// TIA Portal V17 program export: 7 tag tables, 61 data types, 15 data blocks, 115 code blocks (in call order from the OBs), 16 instance data blocks

VAR_GLOBAL   // PLC tag table "Auxiliary_IO"
   Rack2Slot20_I AT %I310.0 : "stET200AL_AQ_I";   //    {ExternalAccessible false, ExternalVisible false, ExternalWritable false}
   Rack2Slot21_I AT %I320.0 : "stET200AL_AI";   //    {ExternalAccessible false, ExternalVisible false, ExternalWritable false}
   Rack1Slot9_I AT %I170.0 : "stET200AL_AI";   //    {ExternalAccessible false, ExternalVisible false, ExternalWritable false}
   Rack1Slot8_I AT %I160.0 : "stET200AL_AI";   //    {ExternalAccessible false, ExternalVisible false, ExternalWritable false}
   Rack1Slot7_I AT %I150.0 : "stET200AL_AI";   //    {ExternalAccessible false, ExternalVisible false, ExternalWritable false}
   Rack2Slot25_I AT %I360.0 : "stET200AL_AI";   //    {ExternalAccessible false, ExternalVisible false, ExternalWritable false}
   Rack1Slot5_I AT %I130.0 : "stET200AL_AI";   //    {ExternalAccessible false, ExternalVisible false, ExternalWritable false}
   Rack1Slot4_I AT %I120.0 : "stET200AL_RTD";   //    {ExternalAccessible false, ExternalVisible false, ExternalWritable false}
   Rack1Slot6_I AT %I140.0 : "stET200AL_AI";   //    {ExternalAccessible false, ExternalVisible false, ExternalWritable false}
   Rack2Slot19_I AT %I300.0 : "stET200AL_AI";   //    {ExternalAccessible false, ExternalVisible false, ExternalWritable false}
   Rack1Slot2_I AT %I100.0 : "stET200AL_AI";   //    {ExternalAccessible false, ExternalVisible false, ExternalWritable false}
   Rack2Slot23_I AT %I340.0 : "stET200AL_AI";   //    {ExternalAccessible false, ExternalVisible false, ExternalWritable false}
   Rack2Slot22_I AT %I330.0 : "stET200AL_AI";   //    {ExternalAccessible false, ExternalVisible false, ExternalWritable false}
   Rack1Slot3_I AT %I110.0 : "stET200AL_RTD";   //    {ExternalAccessible false, ExternalVisible false, ExternalWritable false}
   Rack2Slot24_I AT %I350.0 : "stET200AL_AI";   //    {ExternalAccessible false, ExternalVisible false, ExternalWritable false}
   Rack2Slot29_I AT %I400.0 : "stET200AL_AI";   //    {ExternalAccessible false, ExternalVisible false, ExternalWritable false}
   Rack2Slot30_I AT %I410.0 : "stET200AL_AI";   //    {ExternalAccessible false, ExternalVisible false, ExternalWritable false}
   Rack2Slot31_I AT %I420.0 : "stET200AL_AI";   //    {ExternalAccessible false, ExternalVisible false, ExternalWritable false}
   Rack2Slot32_I AT %I430.0 : "stET200AL_RTD";   //    {ExternalAccessible false, ExternalVisible false, ExternalWritable false}
   Rack2Slot33_I AT %I440.0 : "stET200AL_AI";   //    {ExternalAccessible false, ExternalVisible false, ExternalWritable false}
   Rack2Slot34_I AT %I450.0 : "stET200AL_AI";   //    {ExternalAccessible false, ExternalVisible false, ExternalWritable false}
   Rack2Slot26_I AT %I370.0 : "stET200AL_AQ_I";   //    {ExternalAccessible false, ExternalVisible false, ExternalWritable false}
   Rack2Slot27_I AT %I380.0 : "stET200AL_AI";   //    {ExternalAccessible false, ExternalVisible false, ExternalWritable false}
   Rack2Slot28_I AT %I390.0 : "stET200AL_AQ_I";   //    {ExternalAccessible false, ExternalVisible false, ExternalWritable false}
   Rack2Slot20_Q AT %Q310.0 : "stET200AL_AQ";   //    {ExternalAccessible false, ExternalVisible false, ExternalWritable false}
   Rack2Slot21_Q AT %Q320.0 : "stET200AL_AQ";   //    {ExternalAccessible false, ExternalVisible false, ExternalWritable false}
   Rack1Slot10_I AT %I180.0 : "stET200AL_DIQ_I";   //    {ExternalAccessible false, ExternalVisible false, ExternalWritable false}
   Rack1Slot11_I AT %I190.0 : "stET200AL_RTD";   //    {ExternalAccessible false, ExternalVisible false, ExternalWritable false}
   Rack1Slot12_I AT %I200.0 : "stET200AL_AI";   //    {ExternalAccessible false, ExternalVisible false, ExternalWritable false}
   Rack1Slot13_I AT %I210.0 : "stET200AL_AI";   //    {ExternalAccessible false, ExternalVisible false, ExternalWritable false}
   Rack1Slot14_I AT %I248.0 : "stET200AL_RTD";   //    {ExternalAccessible false, ExternalVisible false, ExternalWritable false}
   Rack1Slot15_I AT %I230.0 : "stET200AL_AI";   //    {ExternalAccessible false, ExternalVisible false, ExternalWritable false}
   Rack1Slot16_I AT %I240.0 : "stET200AL_AI";   //    {ExternalAccessible false, ExternalVisible false, ExternalWritable false}
   Rack1Slot17_I AT %I250.0 : "stET200AL_AI";   //    {ExternalAccessible false, ExternalVisible false, ExternalWritable false}
   Rack2Slot19_Q AT %Q300.0 : "stET200AL_AQ";   //    {ExternalAccessible false, ExternalVisible false, ExternalWritable false}
   Rack2Slot22_Q AT %Q330.0 : "stET200AL_AQ";   //    {ExternalAccessible false, ExternalVisible false, ExternalWritable false}
   Rack2Slot23_Q AT %Q340.0 : "stET200AL_AQ";   //    {ExternalAccessible false, ExternalVisible false, ExternalWritable false}
   Rack2Slot24_Q AT %Q350.0 : "stET200AL_AQ";   //    {ExternalAccessible false, ExternalVisible false, ExternalWritable false}
   Rack2Slot25_Q AT %Q360.0 : "stET200AL_AQ";   //    {ExternalAccessible false, ExternalVisible false, ExternalWritable false}
   Rack2Slot26_Q AT %Q370.0 : "stET200AL_AQ";   //    {ExternalAccessible false, ExternalVisible false, ExternalWritable false}
   Rack2Slot27_Q AT %Q380.0 : "stET200AL_AQ";   //    {ExternalAccessible false, ExternalVisible false, ExternalWritable false}
   Rack2Slot28_Q AT %Q390.0 : "stET200AL_AQ";   //    {ExternalAccessible false, ExternalVisible false, ExternalWritable false}
   Rack2Slot29_Q AT %Q400.0 : "stET200AL_AQ";   //    {ExternalAccessible false, ExternalVisible false, ExternalWritable false}
   Rack2Slot30_Q AT %Q410.0 : "stET200AL_AQ";   //    {ExternalAccessible false, ExternalVisible false, ExternalWritable false}
   Rack2Slot31_Q AT %Q420.0 : "stET200AL_AQ";   //    {ExternalAccessible false, ExternalVisible false, ExternalWritable false}
   Rack2Slot32_Q AT %Q430.0 : "stET200AL_AQ";   //    {ExternalAccessible false, ExternalVisible false, ExternalWritable false}
   Rack2Slot33_Q AT %Q440.0 : "stET200AL_AQ";   //    {ExternalAccessible false, ExternalVisible false, ExternalWritable false}
   Rack2Slot34_Q AT %Q450.0 : "stET200AL_AQ";   //    {ExternalAccessible false, ExternalVisible false, ExternalWritable false}
   Rack1Slot10_Q AT %Q180.0 : "stET200AL_DIQ_Q";   //    {ExternalAccessible false, ExternalVisible false, ExternalWritable false}
END_VAR

VAR_GLOBAL   // PLC tag table "Default tag table"
   Trial AT %I0.0 : Bool;
END_VAR

VAR_GLOBAL   // PLC tag table "Inverters"
   TA1_Rx AT %I10.0 : "stABB_ACSx80_Rx";   // HBL-SC-01   {ExternalAccessible false, ExternalVisible false, ExternalWritable false}
   TA1_Tx AT %Q10.0 : "stABB_ACSx80_Tx";   // HBL-SC-01   {ExternalAccessible false, ExternalVisible false, ExternalWritable false}
   TA2_Rx AT %I30.0 : "stABB_ACSx80_Rx";   // HBL-SC-02   {ExternalAccessible false, ExternalVisible false, ExternalWritable false}
   TA10_Rx AT %I68.0 : "stABB_ACSx80_Rx";   // HBL-SC-10   {ExternalAccessible false, ExternalVisible false, ExternalWritable false}
   TA2_Tx AT %Q30.0 : "stABB_ACSx80_Tx";   // HBL-SC-02   {ExternalAccessible false, ExternalVisible false, ExternalWritable false}
   TA10_Tx AT %Q68.0 : "stABB_ACSx80_Tx";   // '   {ExternalAccessible false, ExternalVisible false, ExternalWritable false}
   TA_State AT %IB7 : Byte;   // 1 = online   {ExternalAccessible false, ExternalVisible false, ExternalWritable false}
   TA3_Rx AT %I228.0 : "stABB_ACSx80_Rx";   // HBL-SC-03   {ExternalAccessible false, ExternalVisible false, ExternalWritable false}
   TA3_Tx AT %Q88.0 : "stABB_ACSx80_Tx";   // HBL-SC-03   {ExternalAccessible false, ExternalVisible false, ExternalWritable false}
END_VAR

VAR_GLOBAL   // PLC tag table "Local_IO"
   SM1222_DO_0 AT %Q8.0 : Bool;   //    {ExternalAccessible false, ExternalVisible false, ExternalWritable false}
   SM1222_DO_1 AT %Q8.1 : Bool;   //    {ExternalAccessible false, ExternalVisible false, ExternalWritable false}
   SM1222_DO_2 AT %Q8.2 : Bool;   //    {ExternalAccessible false, ExternalVisible false, ExternalWritable false}
   SM1222_DO_3 AT %Q8.3 : Bool;   //    {ExternalAccessible false, ExternalVisible false, ExternalWritable false}
   SM1222_DO_4 AT %Q8.4 : Bool;   //    {ExternalAccessible false, ExternalVisible false, ExternalWritable false}
   SM1222_DO_5 AT %Q8.5 : Bool;   //    {ExternalAccessible false, ExternalVisible false, ExternalWritable false}
   SM1222_DO_6 AT %Q8.6 : Bool;   //    {ExternalAccessible false, ExternalVisible false, ExternalWritable false}
   SM1222_DO_7 AT %Q8.7 : Bool;   //    {ExternalAccessible false, ExternalVisible false, ExternalWritable false}
   SM531 AT %I500.0 : "stSM531_4AI";   //    {ExternalAccessible false, ExternalVisible false, ExternalWritable false}
   SM521 AT %I510.0 : "stSM521_16DI";   //    {ExternalAccessible false, ExternalVisible false, ExternalWritable false}
   SM522_I AT %I512.0 : "stSM522_32DQ_I";   //    {ExternalAccessible false, ExternalVisible false, ExternalWritable false}
   SM522_Q AT %Q512.0 : "stSM522_32DQ_Q";   //    {ExternalAccessible false, ExternalVisible false, ExternalWritable false}
END_VAR

VAR_GLOBAL   // PLC tag table "RIO1"
   RIO1_Slot4_I AT %I634.0 : "stSM531_8AI";   //    {ExternalAccessible false, ExternalVisible false, ExternalWritable false}
   RIO1_Slot2_I AT %I600.0 : "stSM531_8AI";   //    {ExternalAccessible false, ExternalVisible false, ExternalWritable false}
   RIO1_Slot3_I AT %I617.0 : "stSM531_8AI";   //    {ExternalAccessible false, ExternalVisible false, ExternalWritable false}
   RIO1_Slot5_I AT %I651.0 : "stSM531_8AI";   //    {ExternalAccessible false, ExternalVisible false, ExternalWritable false}
   RIO1_Slot6_I AT %I668.0 : "stSM531_8AI";   //    {ExternalAccessible false, ExternalVisible false, ExternalWritable false}
   RIO1_Slot7_I AT %I685.0 : "stSM531_8AI";   //    {ExternalAccessible false, ExternalVisible false, ExternalWritable false}
   RIO1_Slot8_I AT %I702.0 : "stSM531_8AI";   //    {ExternalAccessible false, ExternalVisible false, ExternalWritable false}
   RIO1_Slot9_I AT %I719.0 : "stSM531_8AI";   //    {ExternalAccessible false, ExternalVisible false, ExternalWritable false}
   RIO1_Slot10_I AT %I736.0 : "stSM531_8AI";   //    {ExternalAccessible false, ExternalVisible false, ExternalWritable false}
   RIO1_Slot11_I AT %I753.0 : "stSM531_8AI";   //    {ExternalAccessible false, ExternalVisible false, ExternalWritable false}
   RIO1_Slot12_I AT %I770.0 : "stSM531_8AI";   //    {ExternalAccessible false, ExternalVisible false, ExternalWritable false}
   RIO1_Slot13_I AT %I787.0 : "stSM521_16DI";   //    {ExternalAccessible false, ExternalVisible false, ExternalWritable false}
   RIO1_Slot14_I AT %I789.0 : "stSM531_8AQ_I";   //    {ExternalAccessible false, ExternalVisible false, ExternalWritable false}
   RIO1_Slot15_I AT %I790.0 : "stSM531_8AQ_I";   //    {ExternalAccessible false, ExternalVisible false, ExternalWritable false}
   RIO1_Slot16_I AT %I791.0 : "stSM522_32DQ_I";   //    {ExternalAccessible false, ExternalVisible false, ExternalWritable false}
   RIO1_Slot14_Q AT %Q600.0 : "stSM531_8AQ";   //    {ExternalAccessible false, ExternalVisible false, ExternalWritable false}
   RIO1_Slot15_Q AT %Q616.0 : "stSM531_8AQ";   //    {ExternalAccessible false, ExternalVisible false, ExternalWritable false}
   RIO1_Slot16_Q AT %Q632.0 : "stSM522_32DQ_Q";   //    {ExternalAccessible false, ExternalVisible false, ExternalWritable false}
END_VAR

VAR_GLOBAL   // PLC tag table "RIO2"
   RIO2_Slot4_I AT %I934.0 : "stSM531_8AI";   //    {ExternalAccessible false, ExternalVisible false, ExternalWritable false}
   RIO2_Slot2_I AT %I900.0 : "stSM531_8AI";   //    {ExternalAccessible false, ExternalVisible false, ExternalWritable false}
   RIO2_Slot3_I AT %I917.0 : "stSM531_8AI";   //    {ExternalAccessible false, ExternalVisible false, ExternalWritable false}
   RIO2_Slot5_I AT %I951.0 : "stSM531_8AI";   //    {ExternalAccessible false, ExternalVisible false, ExternalWritable false}
   RIO2_Slot6_I AT %I968.0 : "stSM531_8AI";   //    {ExternalAccessible false, ExternalVisible false, ExternalWritable false}
   RIO2_Slot7_I AT %I985.0 : "stSM531_8AI";   //    {ExternalAccessible false, ExternalVisible false, ExternalWritable false}
   RIO2_Slot8_I AT %I1002.0 : "stSM531_8AI";   //    {ExternalAccessible false, ExternalVisible false, ExternalWritable false}
   RIO2_Slot9_I AT %I1019.0 : "stSM531_8AI";   //    {ExternalAccessible false, ExternalVisible false, ExternalWritable false}
   RIO2_Slot10_I AT %I1036.0 : "stSM531_8AI";   //    {ExternalAccessible false, ExternalVisible false, ExternalWritable false}
   RIO2_Slot11_I AT %I1053.0 : "stSM531_8AI";   //    {ExternalAccessible false, ExternalVisible false, ExternalWritable false}
   RIO2_Slot12_I AT %I1070.0 : "stSM531_8AI";   //    {ExternalAccessible false, ExternalVisible false, ExternalWritable false}
   RIO2_Slot13_I AT %I1087.0 : "stSM521_16DI";   //    {ExternalAccessible false, ExternalVisible false, ExternalWritable false}
   RIO2_Slot14_I AT %I1089.0 : "stSM531_8AQ_I";   //    {ExternalAccessible false, ExternalVisible false, ExternalWritable false}
   RIO2_Slot15_I AT %I1090.0 : "stSM531_8AQ_I";   //    {ExternalAccessible false, ExternalVisible false, ExternalWritable false}
   RIO2_Slot16_I AT %I1091.0 : "stSM522_32DQ_I";   //    {ExternalAccessible false, ExternalVisible false, ExternalWritable false}
   RIO2_Slot14_Q AT %Q900.0 : "stSM531_8AQ";   //    {ExternalAccessible false, ExternalVisible false, ExternalWritable false}
   RIO2_Slot15_Q AT %Q916.0 : "stSM531_8AQ";   //    {ExternalAccessible false, ExternalVisible false, ExternalWritable false}
   RIO2_Slot16_Q AT %Q932.0 : "stSM522_32DQ_Q";   //    {ExternalAccessible false, ExternalVisible false, ExternalWritable false}
END_VAR

VAR_GLOBAL   // PLC tag table "Standard-Variable-Table"
   Clock_Byte AT %MB0 : Byte;   //    {ExternalAccessible false, ExternalVisible false, ExternalWritable false}
   Clock_10Hz AT %M0.0 : Bool;   //    {ExternalAccessible false, ExternalVisible false, ExternalWritable false}
   Clock_5Hz AT %M0.1 : Bool;   //    {ExternalAccessible false, ExternalVisible false, ExternalWritable false}
   "Clock_2.5Hz" AT %M0.2 : Bool;   //    {ExternalAccessible false, ExternalVisible false, ExternalWritable false}
   Clock_2Hz AT %M0.3 : Bool;   //    {ExternalAccessible false, ExternalVisible false, ExternalWritable false}
   "Clock_1.25Hz" AT %M0.4 : Bool;   //    {ExternalAccessible false, ExternalVisible false, ExternalWritable false}
   Clock_1Hz AT %M0.5 : Bool;   //    {ExternalAccessible false, ExternalVisible false, ExternalWritable false}
   "Clock_0.625Hz" AT %M0.6 : Bool;   //    {ExternalAccessible false, ExternalVisible false, ExternalWritable false}
   "Clock_0.5Hz" AT %M0.7 : Bool;   //    {ExternalAccessible false, ExternalVisible false, ExternalWritable false}
   System_Byte AT %MB1 : Byte;   //    {ExternalAccessible false, ExternalVisible false, ExternalWritable false}
   FirstScan AT %M1.0 : Bool;   //    {ExternalAccessible false, ExternalVisible false, ExternalWritable false}
   DiagStatusUpdate AT %M1.1 : Bool;   //    {ExternalAccessible false, ExternalVisible false, ExternalWritable false}
   AlwaysTRUE AT %M1.2 : Bool;   //    {ExternalAccessible false, ExternalVisible false, ExternalWritable false}
   AlwaysFALSE AT %M1.3 : Bool;   //    {ExternalAccessible false, ExternalVisible false, ExternalWritable false}
   CVM1 AT %IW472 : Word;   //    {ExternalAccessible false, ExternalVisible false, ExternalWritable false}
   CVM2 AT %IW474 : Word;   //    {ExternalAccessible false, ExternalVisible false, ExternalWritable false}
   ModbusOK AT %I476.0 : Bool;   //    {ExternalAccessible false, ExternalVisible false, ExternalWritable false}
END_VAR
VAR_GLOBAL CONSTANT   // user constants
   Keiner : Pip := 65535;
   "Automatische Aktualisierung" : Pip := 0;
   "TPA 1" : Pip := 1;
   "TPA 2" : Pip := 2;
   "TPA 3" : Pip := 3;
   "TPA 4" : Pip := 4;
   "TPA OB Servo" : Pip := 32768;
   "Local~MC(1)" : Hw_SubModule := 51;
   "Local~Exec(1)" : Hw_SubModule := 52;
   "Local(1)" : Hw_SubModule := 49;
   "Local~HSC_1" : Hw_Hsc := 257;
   "Local~HSC_2" : Hw_Hsc := 258;
   "Local~HSC_3" : Hw_Hsc := 259;
   "Local~HSC_4" : Hw_Hsc := 260;
   "Local~HSC_5" : Hw_Hsc := 261;
   "Local~HSC_6" : Hw_Hsc := 262;
   "Local~AI_2_AQ_2_1" : Hw_SubModule := 263;
   "Local~DI_14_DQ_10_1" : Hw_SubModule := 264;
   "Local~Pulse_1" : Hw_Pwm := 265;
   "Local~Pulse_2" : Hw_Pwm := 266;
   "Local~Pulse_3" : Hw_Pwm := 267;
   "Local~Pulse_4" : Hw_Pwm := 268;
   Engine1InPosition : Event_HwInt := 16#C0000101;
   HallSensorFlag4 : Event_HwInt := 16#C0050108;
   HallSensorFlag1 : Event_HwInt := 16#C0020108;
   HallSensorFlag2 : Event_HwInt := 16#C0030108;
   HallSensorFlag3 : Event_HwInt := 16#C0040108;
   "Sensors~KF102" : Hw_SubModule := 448;
   "Local~Common(1)" : Hw_SubModule := 50;
   "Local~Device(1)" : Hw_Device := 32;
   "Local~Configuration(1)" : Hw_SubModule := 33;
   "Local~OPC_UA" : Hw_SubModule := 117;
   "OB_Time error interrupt(1)" : OB_TIMEERROR := 80;
   "Local~DQ_8xRelay" : Hw_SubModule := 270;
   "Sensors~KF103" : Hw_SubModule := 278;
   "Sensors~KF104" : Hw_SubModule := 271;
   "Sensors~KF105" : Hw_SubModule := 272;
   "Sensors~KF106" : Hw_SubModule := 274;
   "Sensors~KF107" : Hw_SubModule := 276;
   "Sensors~KF108" : Hw_SubModule := 277;
   "Sensors~KF109" : Hw_SubModule := 279;
   "Sensors~KF110" : Hw_SubModule := 280;
   "Sensors~KF219" : Hw_SubModule := 284;
   "Sensors~KF220" : Hw_SubModule := 285;
   "Sensors~KF221" : Hw_SubModule := 286;
   "Sensors~KF222" : Hw_SubModule := 287;
   "Sensors~KF223" : Hw_SubModule := 288;
   "Sensors~KF224" : Hw_SubModule := 289;
   "Sensors~KF227" : Hw_SubModule := 292;
   "Sensors~KF225" : Hw_SubModule := 293;
   "Sensors~KF226" : Hw_SubModule := 290;
   "Sensors~KF228" : Hw_SubModule := 291;
   "Local~AI_1xRTD_1" : Hw_SubModule := 294;
   "Local~PROFINET_interface_1(1)" : Hw_Interface := 64;
   "Local~PROFINET_interface_1~Port_2(1)" : Hw_Interface := 66;
   "Local~PROFINET_interface_1~Port_1(1)" : Hw_Interface := 65;
   "Local~PROFINET_IO-System" : Hw_IoSystem := 269;
   "Sensors~Proxy" : Hw_SubModule := 441;
   "Sensors~IODevice" : Hw_Device := 275;
   "Sensors~Head" : Hw_SubModule := 442;
   "Sensors~PROFINET_interface" : Hw_Interface := 443;
   "Sensors~PROFINET_interface~Port_1" : Hw_Interface := 444;
   "Sensors~PROFINET_interface~Port_2" : Hw_Interface := 445;
   "Sensors~ET-Con_2" : Hw_SubModule := 449;
   "Sensors~ET-Con_1" : Hw_SubModule := 447;
   "Sensors~KF111" : Hw_SubModule := 281;
   "OB_Main(1)" : OB_PCYCLE := 1;
   "HBL-SC-02~Proxy" : Hw_SubModule := 283;
   "HBL-SC-02~IODevice" : Hw_Device := 273;
   "HBL-SC-02~Interface" : Hw_Interface := 295;
   "HBL-SC-02~Interface~Port_1" : Hw_Interface := 296;
   "HBL-SC-02~Interface~Port_2" : Hw_Interface := 297;
   "HBL-SC-02~Head" : Hw_SubModule := 298;
   "HBL-SC-02~PPO_Type_6_1" : Hw_SubModule := 299;
   "HBL-SC-10~Proxy" : Hw_SubModule := 302;
   "HBL-SC-10~IODevice" : Hw_Device := 300;
   "HBL-SC-10~Interface" : Hw_Interface := 303;
   "HBL-SC-10~Interface~Port_1" : Hw_Interface := 304;
   "HBL-SC-10~Interface~Port_2" : Hw_Interface := 305;
   "HBL-SC-10~Head" : Hw_SubModule := 306;
   "HBL-SC-10~PPO_Type_6_1" : Hw_SubModule := 307;
   "HBL-SC-01~Proxy" : Hw_SubModule := 310;
   "HBL-SC-01~IODevice" : Hw_Device := 308;
   "HBL-SC-01~Interface" : Hw_Interface := 311;
   "HBL-SC-01~Interface~Port_1" : Hw_Interface := 312;
   "HBL-SC-01~Interface~Port_2" : Hw_Interface := 313;
   "HBL-SC-01~Head" : Hw_SubModule := 314;
   "HBL-SC-01~PPO_Type_6_1" : Hw_SubModule := 315;
   "OB_Main_Cyclic(1)" : OB_Cyclic := 30;
END_VAR

TYPE "stPrimerPump"
// stored: IsFailsafeCompliant false
   STRUCT
      fMotorSpeed : Real;   // [rpm] Fixed motor speed
      fMotorTorqueLimit : Real;   // [%] Torque limit
      fOut : Real;   // [rpm]
      Controller : "stOnOffRegulator";
   END_STRUCT;
END_TYPE

TYPE "stProcessValve2"
// stored: IsFailsafeCompliant false
   STRUCT
      bOpenRequest : Bool;   // Auto mode command. 1 = open valve, 0 = do nothing
      bCloseRequest : Bool;   // Auto mode command. 1 = close valve, 0 = do nothing
      bOpenStatus : Bool;   // Feedback from valve. 1 = valve is open, 0 = valve is not open
      bClosedStatus : Bool;   // Feedback from valve. 1 = valve is closed, 0 = valve is not closed
      bNormalState : Bool;   // 1 = Normally Open, 0 = Normally Closed
      bOpenCommand : Bool;   // Output to valve. 1 = drive in oipen direction, 0 = do not drive in open direction
      bCloseCommand : Bool;   // Output to valve. 1 = drive in closed direction, 0 = do not drive in closed direction
      bManualMode : Bool;   // 1 = Manual Mode, 0 = not Manual Mode
      bManualOpenRequest : Bool;   // Manual mode command. 1 = open valve, 0 = do nothing
      bManualCloseRequest : Bool;   // Manual mode command. 1 = close valve, 0 = do nothing
      nState : USInt := 0;   // 0 = unknown, 1 = closed, 2 = opening, 3 = open, 4 = closing, 5 = closing error, 6 = opening error
      tOpeningTimeout : Time := T#5s;   // Time to allow for opening before flagging an error
      tClosingTimeout : Time := T#5s;   // Time to allow for closing before flagging an error
   END_STRUCT;
END_TYPE

TYPE "stProfile"
// stored: IsFailsafeCompliant false
   STRUCT
      lfMemory : LReal;   // Internal state
      lfElapsed : LReal;   // Profile value
   END_STRUCT;
END_TYPE

TYPE "typeDataPtr"
// stored: IsFailsafeCompliant false
   STRUCT
      data : Array[0..7] of Word;
   END_STRUCT;
END_TYPE

TYPE "stAlarmState"
// stored: IsFailsafeCompliant false
   STRUCT
      bActive : Bool;   // 1 = active, 0 = not active
      bActiveUnack : Bool;   // 1 = unacknowledged, 0 = acknowledged
      bAck : Bool;   // 1 = acknowledge (pulse signal)
   END_STRUCT;
END_TYPE

TYPE "stDeviationAlarm"
// stored: IsFailsafeCompliant false
   STRUCT
      bEnable : Bool := true;   // 1 = enable, 0 = block
      fDeviationLimit : Real;   // Alarm threshold
      tActivationDelay : Time;   // Alarm activation delay
      sState : "stAlarmState";   // Alarm
   END_STRUCT;
END_TYPE

TYPE "stDigitalAlarm"
// stored: IsFailsafeCompliant false
   STRUCT
      bEnable : Bool := true;   // 1 = enabled, 0 = blocked
      bInput : Bool;   // 1 = active, 0 = not active
      tActivationDelay : Time;   // Alarm activation delay
      sState : "stAlarmState";   // Alarm
   END_STRUCT;
END_TYPE

TYPE "stEvent"
// stored: IsFailsafeCompliant false
   STRUCT
      bEnable : Bool := true;   // 1 = enable, 0 = block
      bInput : Bool;   // 1 = active, 0 = not active
      sState : "stAlarmState";   // Alarm
   END_STRUCT;
END_TYPE

TYPE "stLimitAlarm"
// stored: IsFailsafeCompliant false
   STRUCT
      bEnable : Bool := true;
      fLimit : Real;   // Alarm threshold
      fHysteresis : Real;   // Deadband around the threshold
      tActivationDelay : Time;   // Alarm activation delay
      sState : "stAlarmState";   // Alarm
   END_STRUCT;
END_TYPE

TYPE "stWinCCAlarm"
// stored: IsFailsafeCompliant false
   STRUCT
      Memory : Int;   // Alarm state
   END_STRUCT;
END_TYPE

TYPE "stCalcSelect"
// stored: IsFailsafeCompliant false
   STRUCT
      nMode : USInt;   // Requested mode (0 = none, 1 = A, 2 = B, 3 = MIN, 4 = MAX, 5 = AVG)
      nActualMode : USInt;   // Actual mode (differs from nMode if bWarning is true)
      bError : Bool;   // 1 = not able to emit any output value, 0 = value ok
      bWarning : Bool;   // 1 = not able to emit requested value, 0 = value ok
   END_STRUCT;
END_TYPE

TYPE "stABB_ACSx80_Rx"
// stored: IsFailsafeCompliant false
   STRUCT
      SW : Word;   // Status Word (58.109)
      Act1 : Word;   // Actual value 1 (58.110)
      Act2 : Word;   // Actual value 2 (58.111)
      DataIO_12 : Word;   // User configurable 1 (58.112)
      DataIO_13 : Word;   // User configurable 2 (58.113)
      DataIO_14 : Word;   // User configurable 3 (58.114)
      DataIO_15 : Word;   // User configurable 4 (58.115)
      DataIO_16 : Word;   // User configurable 5 (58.116)
   END_STRUCT;
END_TYPE

TYPE "stABB_ACSx80_Tx"
// stored: IsFailsafeCompliant false
   STRUCT
      CW : Word;   // Command word (58.101)
      Ref1 : Word;   // Reference 1 (58.102)
      Ref2 : Word;   // Reference 2 (58.103)
      DataIO_4 : Word;   // User configurable 1 (58.104)
      DataIO_5 : Word;   // User configurable 2 (58.105)
      DataIO_6 : Word;   // User configurable 3 (58.106)
      DataIO_7 : Word;   // User configurable 4 (58.107)
      DataIO_8 : Word;   // User configurable 5 (58.108)
   END_STRUCT;
END_TYPE

TYPE "stHeartbeat"
// stored: IsFailsafeCompliant false
   STRUCT
      bOut : Bool;   // Bit sent to remote partner
      bIn : Bool;   // Bit received from remote partner
      bEnable : Bool;   // 1 = run heartbeat, 0 = disabled
      bOk : Bool;   // 1 = heatbeat ok, 0 = timeout
      nState : USInt;   // Heartbeat state
      tTimeout : Time;   // Timeout before comm error
   END_STRUCT;
END_TYPE

TYPE "stHeartbeatCount2"
// stored: IsFailsafeCompliant false
   STRUCT
      nLocalCount : UInt;   // Count sent to remote partner
      nRemoteCount : UInt;   // Count received from remote partner
      bEnable : Bool;   // 1 = run heartbeat, 0 = disabled
      bOk : Bool;   // 1 = heatbeat ok, 0 = timeout
      nState : USInt;   // 0 = idle, 1 = ping, 2 = wait for pong, 3 = timeout
      tTimeout : Time := T#2s;   // Comm error timeout
   END_STRUCT;
END_TYPE

TYPE "stHoursCounter"
// stored: IsFailsafeCompliant false
   STRUCT
      nHours : UDInt;   // 0-4294967295
      nMinutes : USInt;   // 0-59
      nSeconds : USInt;   // 0-59
      bReset : Bool;   // Command bit to reset the count
   END_STRUCT;
END_TYPE

TYPE "stCirculationPump"
// stored: IsFailsafeCompliant false
   STRUCT
      bEnable : Bool;   // 1 = enabled 0 = disabled
      bManualMode : Bool;   // 1 = manual, 0 = auto
      bManualRun : Bool;   // 1 = force run, 0 = off
      bOutput : Bool;   // 1 = run, 0 = stop
      bFault : Bool;   // 1 = fault, 0 = ok
      bPressureLow : Bool;   // 1 = pressure low, 0 = ok
      bTemperatureHigh : Bool;   // 1 = temperature high, 0 = ok
      bDifferentialPressureHigh : Bool;   // 1 = pressure high, 0 = ok
      bReservoirLow : Bool;   // 1 = reservoir low, 0 = ok
      bDeltaTHigh : Bool;   // 1 = delta T high, 0 = ok
      bPressureHigh : Bool;   // 1 = pressure high, 0 = ok
      nMode : USInt;   // 0 = Off, 1 = Auto, 2 = Manual
   END_STRUCT;
END_TYPE

TYPE "stFilterDryer"
// stored: IsFailsafeCompliant false
   STRUCT
      fFixedOutput : Real;   // Value to set output to when active
      fOut : Real;   // Controller output
      Controller : "stPeriodicRegulator";
   END_STRUCT;
END_TYPE

TYPE "stNullRegulator"
// stored: IsFailsafeCompliant false
   STRUCT
      bEnable : Bool;   // 1 = regulator on, 0 = regulator off
      fSetpoint : Real;   // Setpoint
      fOutMax : Real;
      fOutMin : Real;
      fOut : Real;   // Manipulated value
      bManualMode : Bool;   // 1 = manual mode, 0 = auto
      fManualValue : Real;
      bAtMin : Bool;   // Controller negative saturation
      bAtMax : Bool;   // Controller positive saturation
      bFault : Bool;   // 1 = controller fault, 0 = ok
      nMode : USInt;   // 0 = Off, 1 = Auto, 2 = Manual
   END_STRUCT;
END_TYPE

TYPE "stOilHeater"
// stored: IsFailsafeCompliant false
   STRUCT
      fOilSuperheat : Real;   // Margin above condensing temperature
      bUseGroup2 : Bool;   // Use Group 2 heaters also
      Controller : "stOnOffRegulator";   // Threshold controller
   END_STRUCT;
END_TYPE

TYPE "stOilRecovery"
// stored: IsFailsafeCompliant false
   STRUCT
      bEnable : Bool;   // Run signal. 1 = Run, 0 = do not run
      nRunRatio : UInt;   // Run once every X times Run signal is active
      fFixedOutput : Real;   // [%] Valve setting when active
      fOut : Real;   // [%] Actual output
      Controller : "stOneShotRegulator";
   END_STRUCT;
END_TYPE

TYPE "stOilSeparator"
// stored: IsFailsafeCompliant false
   STRUCT
      Stage1 : "stOnOffRegulator2";
      Stage2 { S7_SetPoint := 'True'} : "stOnOffRegulator2";
   END_STRUCT;
END_TYPE

TYPE "stOnOffRegulator"
// stored: IsFailsafeCompliant false
   STRUCT
      bEnable : Bool;   // 1 = controller enabled, 0 = disabled
      fSetpoint : Real;   // Controller setpoint
      fHysteresis : Real := 0.5;   // Deadband around setpoint
      bOutput : Bool;   // 1 = output active
      bAtSetpoint : Bool;   // 1 = at setpoint
      bManualMode : Bool;   // 1 = activate manual mode
      fManualSetpoint : Real;   // Manual controller setpoint
      bManualOverride : Bool;   // 1 = activate override
      bOverrideCmd : Bool;   // 1 = force output on
      bFault : Bool;   // 1 = controller fault, 0 = ok
      nMode : USInt;   // 0 = Off, 1 = Auto, 2 = Manual, 3 = Manual Override
   END_STRUCT;
END_TYPE

TYPE "stOnOffRegulator2"
// stored: IsFailsafeCompliant false
   STRUCT
      bEnable : Bool;   // 1 = controller enabled, 0 = disabled
      bOutput : Bool;   // 1 = output active
      bAtSetpoint : Bool;   // 1 = at setpoint
      bManualOverride : Bool;   // 1 = activate override
      bOverrideCmd : Bool;   // 1 = force output on
      bFault : Bool;   // 1 = controller fault, 0 = ok
      nMode : USInt;   // 0 = Off, 1 = Auto, 2 = Manual, 3 = Manual Override
   END_STRUCT;
END_TYPE

TYPE "stOnOffRegulator3"
// stored: IsFailsafeCompliant false
   STRUCT
      bEnable : Bool;   // 1 = controller enabled, 0 = disabled
      bOutput : Bool;   // 1 = output active
      bAtSetpoint : Bool;   // 1 = at setpoint
      bManualOverride : Bool;   // 1 = activate override
      bOverrideCmd : Bool;   // 1 = force output on
      bFault : Bool;   // 1 = controller fault, 0 = ok
      nMode : USInt;   // 0 = Off, 1 = Auto, 2 = Manual, 3 = Manual Override
      nActivationTime : Time;   // Time to stay active when triggered
   END_STRUCT;
END_TYPE

TYPE "stOneShotRegulator"
// stored: IsFailsafeCompliant false
   STRUCT
      bEnable : Bool;   // 1 = controller enabled, 0 = disabled
      bFault : Bool;   // 1 = controller fault, 0 = ok
      bReset : Bool;   // 1 = reset manual modes, 0 = do nothing
      nMode : USInt;   // 0 = Off, 1 = Auto, 2 = Manual, 3 = Manual Override
      bOutput : Bool;   // 1 = output active
      tOnTime : Time;   // Active time
      tStartDelay : Time;   // Time offset before triggering
      tOnTimeElapsed : Time;   // Elapsed time
      tStartDelayElapsed : Time;   // Elapsed time
      bManualOverride : Bool;   // 1 = activate override
      bOverrideCmd : Bool;   // 1 = force output on
   END_STRUCT;
END_TYPE

TYPE "stPID_Regulator"
// stored: IsFailsafeCompliant false
   STRUCT
      fControlDeviation : Real;   // Deviation = SP - PV
      fOutMax : Real;
      fOutMin : Real;
      fOut : Real;   // Manipulated value
      bManualMode : Bool;   // 1 = manual mode, 0 = auto
      fManualValue : Real;
      Kp : Real;   // Proportional gain
      Tn : Real;   // Integral gain (reset time)
      Tv : Real;   // Velocity or derivative gain
      T1 : Real;   // Differentiator smoothing factor
      bAtMin : Bool;   // Controller negative saturation
      bAtMax : Bool;   // Controller positive saturation
   END_STRUCT;
END_TYPE

TYPE "stPID_Regulator_neu"
// stored: IsFailsafeCompliant false
   STRUCT
      fControlDeviation : Real;   // Deviation = SP - PV
      fFeedbackHysteresis : Real;
      fOutMax : Real;
      fOutMin : Real;
      fOut : Real;   // Manipulated value
      bManualMode : Bool;   // 1 = manual mode, 0 = auto
      fManualValue : Real;
      Kp : Real;   // Proportional gain
      Tn : Real;   // Integral gain (reset time)
      Tv : Real;   // Velocity or derivative gain
      T1 : Real;   // Pixie dust gain
      bAtMin : Bool;   // Controller negative saturation
      bAtMax : Bool;   // Controller positive saturation
   END_STRUCT;
END_TYPE

TYPE "stPIP_Regulator"
TITLE = Position-velocity controller
// Cascaded PI-P form
// stored: IsFailsafeCompliant false
   STRUCT
      bEnable : Bool;   // 1 = regulator on, 0 = regulator off
      fPV : Real;   // Process value (position)
      fPVvel : Real;   // Process value (velocity)
      fSP : Real;   // Setpoint (position)
      fOutMax : Real;   // Max regulator output
      fOutMin : Real;   // Min regulator output
      fVelMax : Real;   // Max velocity
      fVelMin : Real;   // Min velocity
      fOut : Real;   // Regulator output
      bManualMode : Bool;   // 1 = manual mode, 0 = auto
      fManualValue : Real;
      Kp : Real;   // Proportional gain (position)
      Tn : Real;   // Integral gain (reset time) (position)
      KpVel : Real;   // Proportional gain (velocity)
      TnVel : Real;   // Integral gain (velocity)
      fFeedbackHysteresis : Real;   // Deadband for velocity integrator
      bAtMin : Bool;   // Regulator output negative saturation
      bAtMax : Bool;   // Regulator output positive saturation
      bFault : Bool;   // 1 = regulator fault, 0 = ok
      nMode : USInt;   // 0 = Off, 1 = Auto, 2 = Manual
   END_STRUCT;
END_TYPE

TYPE "stPI_Regulator"
// stored: IsFailsafeCompliant false
   STRUCT
      bEnable : Bool;   // 1 = regulator on, 0 = regulator off
      fPV : Real;   // Process value
      fSP : Real;   // Setpoint
      fOutMax : Real;
      fOutMin : Real;
      fOut : Real;   // Manipulated value
      bManualMode : Bool;   // 1 = manual mode, 0 = auto
      fManualValue : Real;
      Kp : Real;   // Proportional gain
      Tn : Real;   // Integral gain (reset time)
      bAtMin : Bool;   // Controller negative saturation
      bAtMax : Bool;   // Controller positive saturation
      bFault : Bool;   // 1 = controller fault, 0 = ok
      nMode : USInt;   // 0 = Off, 1 = Auto, 2 = Manual
   END_STRUCT;
END_TYPE

TYPE "stPerformanceControl"
// stored: IsFailsafeCompliant false
   STRUCT
      RunningCondition : Bool;   // 1 = motor run, 0 = motor stop
      RestrictionID : Int;   // Currently active restriction
      TargetValue : Real;   // Currently selected setpoint [C]
      CurrentValue : Real;   // Currently selected process value [C]
      fOut : Real;   // Compressor performance setpoint [%]
      Settings : "PerformanceControl-STRUCT";
      ManualMode : Struct
         ForceMaxPower : Bool;
         ForceMaxPowerAll : Bool;
         ForcePowerSetpoint : Bool;
         ForcePowerSetpointValue : Real;
      END_STRUCT;
   END_STRUCT;
   // // Settings.SwitchToStandby_timeDelay : Time until MinimumPerformnceRate leads to standby
END_TYPE

TYPE "stPeriodicRegulator"
// stored: IsFailsafeCompliant false
   STRUCT
      bEnable : Bool;   // 1 = controller enabled, 0 = disabled
      bFault : Bool;   // 1 = controller fault, 0 = ok
      bReset : Bool;   // 1 = reset manual modes, 0 = do nothing
      nMode : USInt;   // 0 = Off, 1 = Auto, 2 = Manual, 3 = Manual Override
      bOutput : Bool;   // 1 = output active
      tOnTime : Time;   // Active time
      tPeriod : Time;   // Repetition time
      tOnTimeElapsed : Time;   // Elapsed time
      tPeriodElapsed : Time;   // Elapsed time
      bManualOverride : Bool;   // 1 = activate override
      bOverrideCmd : Bool;   // 1 = force output on
   END_STRUCT;
END_TYPE

TYPE "stPeriodicRegulatorFixed"
// stored: IsFailsafeCompliant false
   STRUCT
      fFixedOutput : Real;   // Value to set output to when active
      fOut : Real;   // Controller output
      Controller : "stPeriodicRegulator";
   END_STRUCT;
END_TYPE

TYPE "stPinchControl"
// stored: IsFailsafeCompliant false
   STRUCT
      bEnable : Bool;   // 1 = enable from HMI, 0 = disable from HMI
      bFault : Bool;   // 1 = fault, 0 = ok
      nMode : USInt;   // 0 = offline, 1 = auto, 2 = manual
      fSetpoint : Real;   // Selected setpoint
      fPV : Real;   // Process value
      Regulator : "stPID_Regulator";
   END_STRUCT;
END_TYPE

TYPE "stProgressivePeriodicRegulator4"
// stored: IsFailsafeCompliant false
   STRUCT
      bEnable : Bool;   // 1 = controller enabled, 0 = disabled
      bFault : Bool;   // 1 = controller fault, 0 = ok
      bOutput : Bool;   // 1 = output active
      bManualOverride : Bool;   // 1 = activate override
      bOverrideCmd : Bool;   // 1 = force output on
      bManualMode : Bool;   // 1 = activate manual mode
      nMode : USInt;   // 0 = Off, 1 = Auto, 2 = Manual, 3 = Manual Override
      tManualPeriod : Time;   // Fixed period
      tOnTime : Time;   // On time of period (duty cycle)
      tPeriod : Time;   // Total period (frequency)
      tOnTimeElapsed : Time;
      tPeriodElapsed : Time;
      fPV : Real;   // Process value
      fPumpSpeed : Real;   // [rpm] Fixed pump speed (hack)
      Param : Struct
         Limit : Array[0..3] of Real;   // Process value thresholds
         Period : Array[0..3] of Time;   // Periods between activations
      END_STRUCT;
   END_STRUCT;
END_TYPE

TYPE "stPurgeControl"
// stored: IsFailsafeCompliant false
   STRUCT
      nPurgeCycles : Int;   // [1] How many purge cycles to run
      nPurgeCyclesRemaining : Int;   // [1] How many purge cycles are left to run
      bEnable : Bool;   // 1 = enable from HMI, 0 = disable from HMI
      bFault : Bool;   // 1 = controller fault, 0 = ok
      bReset : Bool;   // 1 = reset controller, 0 = do nothing
      bPurging : Bool;   // 1 = purging, 0 = not purging
      bSpinning : Bool;   // 1 = spinning, 0 = not spinning
      bDone : Bool;   // 1 = purge cycle completed, 0 = not completed
      nMode : USInt;   // 0 = off, 1 = auto, 2 = manual
      fSpinOut : Real;   // [rpm] Spin setpoint (includes ramping)
      Purge : Struct
         nPurgeType : USInt;   // 0 = timer, 1 = delta P, 2 = timer or delta P, 3 = no purge
         tPurgeTime : Time;   // [s] How long to open the purge valves
         fPurgeDeltaP : Real;   // [kPa] Lower limit for pump delta P
      END_STRUCT;
      Spin : Struct
         tSpinTime : Time;   // [s] How long to spin for
         fSpinSpeed : Real;   // [rpm] Spin speed
         fSpinRamp : Real;   // [rpm/s] Spin ramp
      END_STRUCT;
   END_STRUCT;
END_TYPE

TYPE "stSuperheatControl"
// stored: IsFailsafeCompliant false
   STRUCT
      bEnable : Bool;   // 1 = enabled from HMI 0 = disabled from HMI
      bFault : Bool;   // 1 = fault 0 = ok
      nMode : USInt;   // 0 = off, 1 = auto, 2 = manual
      Regulator : "stPID_Regulator_neu";
      fineTuningRecTarget : Real;   // Parameter (0-1). Smaller value will lead to higher power and reduces expander inlet temperatures (superheat), but makes it more instable. The factor in front will increase the (relative) impact
      ExponentialPinchFactor : Real;
      AdditionalSuperheat : Real;
      "FORCE!_FixedPinch" : Bool;
      "FORCE!_FixedPinch_Value" : Real;
   END_STRUCT;
   // Regulator.Kp := 1.0;
   // Regulator.Tn := 1.0;
   // Regulator.Tv := 1.0;
END_TYPE

TYPE "stTemperatureController2"
// stored: IsFailsafeCompliant false
   STRUCT
      bEnable : Bool;   // 1 = controller active, 0 = controller inactive
      fHeatingSetpoint : Real;   // When below this temp, begin heating
      fCoolingSetpoint : Real;   // When above this temp, begin cooling
      bHeating : Bool;   // 1 = heating on, 0 = heating off
      bCooling : Bool;   // 1 = cooling on, 0 = cooling off
      bAtSetpoint : Bool;   // 1 = at setpoint, 0 = not at setpoint
      bFault : Bool;   // 1 = controller fault, 0 = ok
      bManualMode : Bool;   // 1 = manual setpoint, 0 = normal
      fManualHeatingSetpoint : Real;
      fManualCoolingSetpoint : Real;
      bManualOverride : Bool;   // 1 = enable forcing outputs
      nOverrideState : USInt;   // 0 = off, 1 = heating, 2 = cooling
      nMode : USInt;   // 0 = Off, 1 = Auto, 2 = Manual, 3 = Manual Override
   END_STRUCT;
END_TYPE

TYPE "stTrackingRegulator"
// stored: IsFailsafeCompliant false
   STRUCT
      bEnable : Bool;   // 1 = controller enabled, 0 = disabled
      fSP : Real;   // Setpoint (eg °C)
      fPV : Real;   // Process value (eg °C)
      fPVvelocity : Real;   // Rate of change of process value (eg °C/sec)
      fOutMax : Real;   // Positive-most manipulated value (eg %)
      fOutMin : Real;   // Negative-most manipulated value (eg %)
      fOut : Real;   // Manipulated value (eg %)
      bManualMode : Bool;   // 1 = manual mode, 0 = auto
      fManualValue : Real;   // Fixed manipulated value (eg %)
      fSlewRatePositive : Real;   // Controller ramp in positive direction (eg %/s)
      fSlewRateNegative : Real;   // Controller ramp in negative direction (eg %/s)
      fHysteresis : Real;   // Deadband around setpoint (eg °C)
      fVelocityPositiveLimit : Real;   // Max positive rate of change of process value (eg °C/s)
      fVelocityNegativeLimit : Real;   // Max negative rate of change of process value (eg °C/s)
      bAtMin : Bool;   // Controller negative saturation
      bAtMax : Bool;   // Controller positive saturation
      bAtSetpoint : Bool;   // Controller within control deadband
      bFault : Bool;   // 1 = controller fault, 0 = ok
      nMode : USInt;   // 0 = Off, 1 = Auto, 2 = Manual
   END_STRUCT;
END_TYPE

TYPE "PerformanceControl-STRUCT"
// stored: IsFailsafeCompliant false
   STRUCT
      MinimumPerformanceRate : Real := 0.0;   // [%]
      SwitchToStandby_timeDelay : Time := T#0s;   // Switches off the engine if the required performance value unterruns minimum perofrmance value for this time. Deactivated if zero
      HeatSink : Struct
         Control_Active : Bool := true;   // 1 = enable controller, 0 = disable controller
         UseFeedFlow : Bool := true;   // 1 = use feed flow, 0 = use return flow
         Setpoint : Real;
         DT_Limit_Standby : Real := 20.0;   // Go to standby
         DT_Limit_Resume : Real := 0.5;   // Resume operation
         Kp : Real := 10.0;   // Proportional gain
         Tn : Real := 60.0;   // Integral gain (reset time)
      END_STRUCT;
      HeatSource : Struct
         Control_Active : Bool := true;   // 1 = enable controller, 0 = disable controller
         UseFeedFlow : Bool := true;   // 1 = use feed flow, 0 = use return flow
         Setpoint : Real;
         DT_Limit_Standby : Real := 40.0;   // Go to standby
         DT_Limit_Resume : Real := 0.5;   // Resume operation
         Kp : Real := 1.0;   // Proportional gain
         Tn : Real := 30.0;   // Integral gain (reset time)
      END_STRUCT;
      VariableControl : Struct
         Control_Active : Bool := true;   // 1 = enable controller, 0 = disable controller
         ReferenceID : USInt := 0;
         Setpoint : Real;
         DT_Limit_Standby : Real := 20.0;   // Go to standby
         DT_Limit_Resume : Real := 10.0;   // Resume operation
         Kp : Real := 1.0;   // Proportional gain
         Tn : Real := 30.0;   // Integral gain (reset time)
      END_STRUCT;
      Config : Struct
         MinimumPerformanceRequirement { S7_SetPoint := 'True'} : Real;   // [%] Below this, additional superheat is required
         MaximumAdditionalSuperheat : Real;   // [C] Superheat to add at MinimumPerformanceRequirement
         INCREASEWITHNORESTRICTION : Real;   // [%/s] Default integrator gain
      END_STRUCT;
   END_STRUCT;
END_TYPE

TYPE "stET200AL_AI"
// stored: IsFailsafeCompliant false
   STRUCT
      CH00 : Int;
      CH01 : Int;
      CH02 : Int;
      CH03 : Int;
      CH00_ok : Bool;
      CH01_ok : Bool;
      CH02_ok : Bool;
      CH03_ok : Bool;
   END_STRUCT;
END_TYPE

TYPE "stET200AL_AQ"
// stored: IsFailsafeCompliant false
   STRUCT
      CH0 : Int;
      CH1 : Int;
      CH2 : Int;
      CH3 : Int;
      Spare : Byte;   // So AI & AQ have the same size
   END_STRUCT;
END_TYPE

TYPE "stET200AL_AQ_I"
// stored: IsFailsafeCompliant false
   STRUCT
      CH00_ok : Bool;
      CH01_ok : Bool;
      CH02_ok : Bool;
      CH03_ok : Bool;
      CH04_ok : Bool;
      CH05_ok : Bool;
      CH06_ok : Bool;
      CH07_ok : Bool;
   END_STRUCT;
END_TYPE

TYPE "stET200AL_DIQ_I"
// stored: IsFailsafeCompliant false
   STRUCT
      DI00 : Bool;
      DI01 : Bool;
      DI02 : Bool;
      DI03 : Bool;
      DI04 : Bool;
      DI05 : Bool;
      DI06 : Bool;
      DI07 : Bool;
      DI08 : Bool;
      DI09 : Bool;
      DI10 : Bool;
      DI11 : Bool;
      DI12 : Bool;
      DI13 : Bool;
      DI14 : Bool;
      DI15 : Bool;
      STAT : Array[0..31] of Bool;   // "Value Status" checked in module parameters
   END_STRUCT;
END_TYPE

TYPE "stET200AL_DIQ_Q"
// stored: IsFailsafeCompliant false
   STRUCT
      DQ00 : Bool;
      DQ01 : Bool;
      DQ02 : Bool;
      DQ03 : Bool;
      DQ04 : Bool;
      DQ05 : Bool;
      DQ06 : Bool;
      DQ07 : Bool;
      DQ08 : Bool;
      DQ09 : Bool;
      DQ10 : Bool;
      DQ11 : Bool;
      DQ12 : Bool;
      DQ13 : Bool;
      DQ14 : Bool;
      DQ15 : Bool;
   END_STRUCT;
END_TYPE

TYPE "stET200AL_RTD"
// stored: IsFailsafeCompliant false
   STRUCT
      CH00 : Int;
      CH01 : Int;
      CH02 : Int;
      CH03 : Int;
      CH00_ok : Bool;
      CH01_ok : Bool;
      CH02_ok : Bool;
      CH03_ok : Bool;
   END_STRUCT;
END_TYPE

TYPE "stSM521_16DI"
// stored: IsFailsafeCompliant false
   STRUCT
      DI00 : Bool;
      DI01 : Bool;
      DI02 : Bool;
      DI03 : Bool;
      DI04 : Bool;
      DI05 : Bool;
      DI06 : Bool;
      DI07 : Bool;
      DI08 : Bool;
      DI09 : Bool;
      DI10 : Bool;
      DI11 : Bool;
      DI12 : Bool;
      DI13 : Bool;
      DI14 : Bool;
      DI15 : Bool;
   END_STRUCT;
END_TYPE

TYPE "stSM522_32DQ_I"
// stored: IsFailsafeCompliant false
   STRUCT
      DQ00_ok : Bool;
      DQ01_ok : Bool;
      DQ02_ok : Bool;
      DQ03_ok : Bool;
      DQ04_ok : Bool;
      DQ05_ok : Bool;
      DQ06_ok : Bool;
      DQ07_ok : Bool;
      DQ08_ok : Bool;
      DQ09_ok : Bool;
      DQ10_ok : Bool;
      DQ11_ok : Bool;
      DQ12_ok : Bool;
      DQ13_ok : Bool;
      DQ14_ok : Bool;
      DQ15_ok : Bool;
      DQ16_ok : Bool;
      DQ17_ok : Bool;
      DQ18_ok : Bool;
      DQ19_ok : Bool;
      DQ20_ok : Bool;
      DQ21_ok : Bool;
      DQ22_ok : Bool;
      DQ23_ok : Bool;
      DQ24_ok : Bool;
      DQ25_ok : Bool;
      DQ26_ok : Bool;
      DQ27_ok : Bool;
      DQ28_ok : Bool;
      DQ29_ok : Bool;
      DQ30_ok : Bool;
      DQ31_ok : Bool;
   END_STRUCT;
END_TYPE

TYPE "stSM522_32DQ_Q"
// stored: IsFailsafeCompliant false
   STRUCT
      DQ00 : Bool;
      DQ01 : Bool;
      DQ02 : Bool;
      DQ03 : Bool;
      DQ04 : Bool;
      DQ05 : Bool;
      DQ06 : Bool;
      DQ07 : Bool;
      DQ08 : Bool;
      DQ09 : Bool;
      DQ10 : Bool;
      DQ11 : Bool;
      DQ12 : Bool;
      DQ13 : Bool;
      DQ14 : Bool;
      DQ15 : Bool;
      DQ16 : Bool;
      DQ17 : Bool;
      DQ18 : Bool;
      DQ19 : Bool;
      DQ20 : Bool;
      DQ21 : Bool;
      DQ22 : Bool;
      DQ23 : Bool;
      DQ24 : Bool;
      DQ25 : Bool;
      DQ26 : Bool;
      DQ27 : Bool;
      DQ28 : Bool;
      DQ29 : Bool;
      DQ30 : Bool;
      DQ31 : Bool;
   END_STRUCT;
END_TYPE

TYPE "stSM531_4AI"
// stored: IsFailsafeCompliant false
   STRUCT
      CH00 : Int;
      CH01 : Int;
      CH02 : Int;
      CH03 : Int;
      CH00_ok : Bool;
      CH01_ok : Bool;
      CH02_ok : Bool;
      CH03_ok : Bool;
   END_STRUCT;
END_TYPE

TYPE "stSM531_8AI"
// stored: IsFailsafeCompliant false
   STRUCT
      CH00 : Int;
      CH01 : Int;
      CH02 : Int;
      CH03 : Int;
      CH04 : Int;
      CH05 : Int;
      CH06 : Int;
      CH07 : Int;
      CH00_ok : Bool;
      CH01_ok : Bool;
      CH02_ok : Bool;
      CH03_ok : Bool;
      CH04_ok : Bool;
      CH05_ok : Bool;
      CH06_ok : Bool;
      CH07_ok : Bool;
   END_STRUCT;
END_TYPE

TYPE "stSM531_8AQ"
// stored: IsFailsafeCompliant false
   STRUCT
      CH00 : Int;
      CH01 : Int;
      CH02 : Int;
      CH03 : Int;
      CH04 : Int;
      CH05 : Int;
      CH06 : Int;
      CH07 : Int;
      Spare : Byte;   // So AI & AQ have the same size
   END_STRUCT;
END_TYPE

TYPE "stSM531_8AQ_I"
// stored: IsFailsafeCompliant false
   STRUCT
      CH00_ok : Bool;
      CH01_ok : Bool;
      CH02_ok : Bool;
      CH03_ok : Bool;
      CH04_ok : Bool;
      CH05_ok : Bool;
      CH06_ok : Bool;
      Ch07_ok : Bool;
   END_STRUCT;
END_TYPE

TYPE "CurrentSetting-STRUCT"
// stored: IsFailsafeCompliant false
   STRUCT
      Fluid { S7_SetPoint := 'True'} : "FluidData-STRUCT";   // Kältemittelspezifische Einstellungen (Wird aus StaticData entnommen)
      Compressor { S7_SetPoint := 'True'} : "CompressorData-STRUCT";   // Kompressorspezifische Einstellungen (Wird aus StaticData entnommen)
      System { S7_SetPoint := 'True'} : "SystemData-STRUCT";   // Systemspezifische Einstellungen (Wird aus StaticData entnommen)
      VariableSetting { S7_SetPoint := 'True'} : "VariableSetting-STRUCT";   // Einstellungen, die über die HMI voreingestellt werden können
      StaticSetting { S7_SetPoint := 'True'} : "StaticSetting-STRUCT";   // Programmparameter um Systemverhalten Abzustimmen
      NewInitialisation_Required : Bool;   // Gets set on configuration changes and reset on restart
      ParameterSet_Ordered : Bool;   // Shows if the parameterset is successfully loaded
      ParameterSet_Indicator : Bool;
      MissingSetting : Struct   // Catch all category. To be sorted.
         Compressor : Struct
            OilPumpCurveCritical : Real := 0.133;   // [kPa/rpm] Minimum adequate oil pump performance
            OilPumpCurveWarning : Real := 0.166;   // [kPa/rpm] Minimum expected oil pump performance
            MinStartupSpeed : Real := 25.0;   // [rpm] Minimum speed at compressor start
            WarmupSpeed : Real := 550.0;   // [rpm] Speed in warmup state
            MinOperationalSpeed : Real := 550.0;   // [rpm] Minimum speed in operation
            MaxOperationalSpeed : Real := 1200.0;   // [rpm] Maximum speed in operation
            OilFilterDeltaPCritical : Real := 150.0;   // [kPa] Maximum oil filter delta P
            OilFilterDeltaPWarning : Real := 100.0;   // [kPa] Warning oil filter delta P
         END_STRUCT;
         System : Struct
            HydrolockSpeed : Real := 330.0;   // [rpm] Max safe speed under hydrolock conditions
            CondenserCoefficient : Real := 13.024;   // [?] Mass flow calculation
            EvaporatorCoefficient : Real := 19.07;   // [?] Mass flow calculation
            SuctionLineDryLimitPressure : Real := 80.0;   // [kPa] Compressor suction pressue when suction line is considered dry
            SuctionLineDryLimitSuperheat : Real := 27.0;   // [C] Compressor suction superheat when suction line is considered dry
            CompressorSuperheatDischargeMinimum : Real := 20.0;   // [C] Lowest permissible compressor discharge superheat in operation
            RecuperatorDeltaTWorking : Real := 3.0;   // [C] Recuperator superheat gain when it is considered working
            RecuperatorDeltaTNotWorking : Real := -2.0;   // [C] Recuperator superheat gain when it is considered not working (can be negative)
            ExpansionValvePositionStart : Real := 5.5;   // [%] Expansion valve position in State 4 Start
            ExpansionValvePositionStartCold : Real := 3.0;   // [%] Expansion valve position in State 4 Start, cold start
            HeatSourceDeltaPFlow : Real := 2.0;   // [kPa] Delta P over the heat source that indicates flow
            HeatSinkDeltaPFlow : Real := 2.0;   // [kPa] Delta P over the heat sink that indicates flow
         END_STRUCT;
         Misc : Struct   // A lot of odds and ends
            CompressorStoppedLimit : Real := 10.0;   // [rpm] Compressor speed at which it is considered stopped
            State2DwellTime { S7_SetPoint := 'True'} : Time := T#10s;   // Standby
            State3DwellTime : Time := T#30s;   // Prepare start
            State4DwellTime : Time := T#30s;   // Start
            State5DwellTime : Time := T#20m;   // Warmup
            State7DwellTime : Time := T#10s;   // Stop
            State2PauseTime : Time := T#10s;   // Minimum pause in standby before resume
            EmergencyStopWaitTime : Time := T#5m;   // Cooldown pause after Emergency stop is reset
            T_HeatSinkTemperatureIn_Max : Real := 75.0;   // [C] Maximum temperature on the suction side of the heat sink
         END_STRUCT;
      END_STRUCT;
   END_STRUCT;
END_TYPE

TYPE "StaticSetting-STRUCT"
// stored: IsFailsafeCompliant false
   STRUCT
      AdditionalSuperHeatOnColdStart { ExternalWritable := 'False'} : Real;
      Limits { ExternalWritable := 'False'} : Struct
         T_Ambient_Max { ExternalWritable := 'False'} : Real := 40.0;
         T_Cabinet_Max { ExternalWritable := 'False'} : Real := 45.0;
      END_STRUCT;
   END_STRUCT;
END_TYPE

TYPE "VariableSetting-STRUCT"
// stored: IsFailsafeCompliant false
   STRUCT
      SystemType : Int;   // Select the used system type
      CompressorType : Int;   // Select the used compressor type
      FluidType : Int;   // Select the used working fluid
      OilPreheating_acv : Bool;   // Activates the oil heaters for pre-heating in state standby
      OilHeatSetpoint_min : Real := 10.0;   // Lowest possible oil heater temperature setpoint
      EnableViaHMI : Bool;   // Allow HMI to start & stop the HB
      EnableViaApplication : Bool;   // Allow the Application PLC to start & stop the HB
      SourceOkFromApplication : Bool;
      SinkOkFromApplication : Bool;
      HeatSourceExternalControl : Bool;   // Heat source auxiliary equipment controlled externally
      HeatSinkExternalControl : Bool;   // Heat sink auxiliary equipment controlled externally
   END_STRUCT;
END_TYPE

TYPE "CompressorData-STRUCT"
// stored: IsFailsafeCompliant false
   STRUCT
      CompressorTypeNumber : Int;
      Limits : Struct   // Kompressor Grenzwerte (Müssen noch definiert werden)
         p_CrankCase_Max : Real;   // kPa
         p_Oil_Min : Real;   // kPa
         n_Compressor_Max : Real;   // RPM
         T_Motor_Max : Real;   // C
         M_Motor_Limit : Real;   // %
         T_Inverter_Max : Real;   // C
      END_STRUCT;
      Constant : Struct   // Kompressor Konstanten (Müssen noch definiert werden)
         CompressionVolume_L : Real;
         CompressionLostPerPressureRatio : Real;
         PumpEfficinecy : Real;
      END_STRUCT;
      Settings : Bool;   // Kompressor Einstellungen (Müssen noch definiert werden)
   END_STRUCT;
END_TYPE

TYPE "FluidBasedLimits-STRUCT"
// stored: IsFailsafeCompliant false
   STRUCT
      T_HeatSourceTemperature_Max : Real;
      T_HeatSourceTemperature_Min : Real;
      T_HeatSinkTemperature_Max : Real;
      T_OilTemperature_Critical : Real := 140.0;
      T_OilSuperheat : Real := 8.0;
      T_CoolingSetpoint : Real := 110.0;
   END_STRUCT;
END_TYPE

TYPE "FluidData-STRUCT"
// stored: IsFailsafeCompliant false
   STRUCT
      "Name" : String;
      FluidTypeNumber : Int;
      SaturationCurve_Temperature_C : Array[0..40] of Real;
      SaturationCurve_Pressure_kPa : Array[0..40] of Real;
      DensityCurve_Pressure_kPa : Array[0..12] of Real;
      DensityCurveLiquide_Densety_kg_m3 : Array[0..12] of Real;
      DensityCurveVapor_Densety_kg_m3 : Array[0..12] of Real;
      DensityCurveVapor_SuperheatCorrection_a : Real;
      DensityCurveVapor_SuperheatCorrection_b : Real;
      EnthalpyMap_Superheat_C : Array[0..8] of Real;
      EnthalpyMap_Pressure_kPa : Array[0..11] of Real;
      EnthalpyMap_Enthalpy_kJ_kg : Array[0..11, 0..8] of Real;
      Limits { S7_SetPoint := 'True'} : "FluidBasedLimits-STRUCT";
      T_AdditionalSuperHeatEvaporator : Real;
      P_CriticalPoint : Real := 99999.9;
   END_STRUCT;
END_TYPE

TYPE "StaticData-STRUCT"
// stored: IsFailsafeCompliant false
   STRUCT
      Fluids { ExternalAccessible := 'False'; ExternalVisible := 'False'; ExternalWritable := 'False'; S7_SetPoint := 'True'} : Array[1..4] of "FluidData-STRUCT";
      CompressorTypes { ExternalAccessible := 'False'; ExternalVisible := 'False'; ExternalWritable := 'False'; S7_SetPoint := 'True'} : Array[1..4] of "CompressorData-STRUCT";
      SystemTypes { ExternalAccessible := 'False'; ExternalVisible := 'False'; ExternalWritable := 'False'; S7_SetPoint := 'True'} : Array[1..6] of "SystemData-STRUCT";
   END_STRUCT;
END_TYPE

TYPE "SystemData-STRUCT"
// stored: IsFailsafeCompliant false
   STRUCT
      SystemTypeNumber : Int;
      Limits : Struct
         T_SuperHeatCompressorIn_Min : Real;
         T_Housing_Max : Real;
         T_CoolingCycle_Max : Real;
         p_CompressorOut_Max : Real;
         p_EvaporatorOut_Max : Real;
      END_STRUCT;
      Constant : Bool;
      Settings : Struct
         CooliungPump_ReversedPWM : Bool;
         MotorCooling_AirFanCooledCycle : Bool;   // True if Air fan cooled otherwiese cooled via heat source cycle. Deactivates oil conditioning/prewarming
         DoubleExpansionValves : Bool;   // If A2 and B2 are present in the system
         Reserve3 : Bool;
         Reserve4 : Bool;
         Reserve5 : Bool;
      END_STRUCT;
   END_STRUCT;
END_TYPE

DATA_BLOCK "DB_AI"   // DB40
{ S7_Optimized_Access := 'FALSE' }
AUTHOR : Heaten
VERSION : 0.1
// stored: AutoNumber true, DBAccessibleFromOPCUA true, DBAccessibleFromWebserver true, IsOnlyStoredInLoadMemory false, IsWriteProtectedInAS false
   VAR RETAIN
      HBL_TT_502 { S7_SetPoint := 'True'} : "stAnalogInput";   // Compressor discharge popoff temperature
      HBL_PT_503 { S7_SetPoint := 'True'} : "stAnalogInput";   // Compressor discharge pressure
      HBL_TT_504 { S7_SetPoint := 'True'} : "stAnalogInput";   // Compressor discharge temperature
      HBL_TT_505 { S7_SetPoint := 'True'} : "stAnalogInput";   // Compressor discharge temperature
      HBL_PT_506 { S7_SetPoint := 'True'} : "stAnalogInput";   // Compressor discharge pressure
      HBL_LT_510 { S7_SetPoint := 'True'} : "stAnalogInput";   // Steam generator condensate level
      HBL_PT_511 { S7_SetPoint := 'True'} : "stAnalogInput";   // Heat sink discharge pressure
      HBL_TT_512 { S7_SetPoint := 'True'} : "stAnalogInput";   // Heat sink discharge temperature
      HBL_TT_516 { S7_SetPoint := 'True'} : "stAnalogInput";   // Steam generator suction temperature
      HBL_PT_517 { S7_SetPoint := 'True'} : "stAnalogInput";   // Steam generator suction pressure
      HBL_TT_518 { S7_SetPoint := 'True'} : "stAnalogInput";   // Heat sink discharge process temperature
      HBL_PT_519 { S7_SetPoint := 'True'} : "stAnalogInput";   // Heat sink discharge process pressure
      HBL_FT_520 { S7_SetPoint := 'True'} : "stAnalogInput";   // Refrigerant flow
      HBL_CT_524 { S7_SetPoint := 'True'} : "stAnalogInput";   // Gas detector steam generator suction popoff
      HBL_TT_525 { S7_SetPoint := 'True'} : "stAnalogInput";   // Steam generator (condenser) suction temperature
      HBL_PT_526 { S7_SetPoint := 'True'} : "stAnalogInput";   // Steam generator (condenser) suction pressure
      HBL_FT_527 { S7_SetPoint := 'True'} : "stAnalogInput";   // Heat sink condensate blowdown flow
      HBL_TT_530 { S7_SetPoint := 'True'} : "stAnalogInput";   // Expansion valve B discharge temperature
      HBL_PT_531 { S7_SetPoint := 'True'} : "stAnalogInput";   // Expansion valve B discharge pressure
      HBL_TT_532 { S7_SetPoint := 'True'} : "stAnalogInput";   // Heat source 1 discharge temperature
      HBL_TT_533 { S7_SetPoint := 'True'} : "stAnalogInput";   // Evaporator 1 discharge temperature
      HBL_PT_534 { S7_SetPoint := 'True'} : "stAnalogInput";   // Evaporator 1 discharge pressure
      HBL_AT_535 { S7_SetPoint := 'True'} : "stAnalogInput";   // Evaporator 1 steam quality
      HBL_CT_538 { S7_SetPoint := 'True'} : "stAnalogInput";   // Gas detector evaporator popoff
      HBL_TT_540 { S7_SetPoint := 'True'} : "stAnalogInput";   // Expansion valve A discharge temperature
      HBL_PT_541 { S7_SetPoint := 'True'} : "stAnalogInput";   // Expansion valve A discharge pressure
      HBL_TT_542 { S7_SetPoint := 'True'} : "stAnalogInput";   // Heat source 2 discharge temperature
      HBL_TT_543 { S7_SetPoint := 'True'} : "stAnalogInput";   // Evaporator 2 discharge temperature
      HBL_PT_544 { S7_SetPoint := 'True'} : "stAnalogInput";   // Evaporator 2 discharge pressure
      HBL_AT_545 { S7_SetPoint := 'True'} : "stAnalogInput";   // Evaporator 2 steam quality
      HBL_TT_546 { S7_SetPoint := 'True'} : "stAnalogInput";   // Heat source suction temperature
      HBL_PT_547 { S7_SetPoint := 'True'} : "stAnalogInput";   // Heast source suction pressure
      HBL_PT_561 { S7_SetPoint := 'True'} : "stAnalogInput";   // Evaporator 1 axis A vacuum pressure
      HBL_PT_562 { S7_SetPoint := 'True'} : "stAnalogInput";   // Evaporator 2 axis A vacuum pressure
      HBL_FT_565 { S7_SetPoint := 'True'} : "stAnalogInput";   // Heat source 1 discharge condensate flow
      HBL_FT_566 { S7_SetPoint := 'True'} : "stAnalogInput";   // Heat source 2 discharge condensate flow
      HBL_TT_571 { S7_SetPoint := 'True'} : "stAnalogInput";   // Compressor suction temperature
      HBL_PT_572 { S7_SetPoint := 'True'} : "stAnalogInput";   // Compressor suction pressure
      HBL_TT_573 { S7_SetPoint := 'True'} : "stAnalogInput";   // Expansion valve suction temperature
      HBL_PT_580 { S7_SetPoint := 'True'} : "stAnalogInput";   // Expansion valve suction pressure
      HBL_LT_610 { S7_SetPoint := 'True'} : "stAnalogInput";   // HP receiver refrigerant level
      HBL_TT_611 { S7_SetPoint := 'True'} : "stAnalogInput";   // Steam generator discharge temperature
      HBL_PT_612 { S7_SetPoint := 'True'} : "stAnalogInput";   // Steam generator discharge pressure
      HBL_CT_615 { S7_SetPoint := 'True'} : "stAnalogInput";   // Gas detector PSV discharge pipe
      HBL_PT_618 { S7_SetPoint := 'True'} : "stAnalogInput";   // HP Receiver pressure
      HBL_CT_620 { S7_SetPoint := 'True'} : "stAnalogInput";   // Gas detector recuperator popoff
      HBL_PT_635 { S7_SetPoint := 'True'} : "stAnalogInput";   // Oil separator stage 1 oil return pressure
      HBL_PT_636 { S7_SetPoint := 'True'} : "stAnalogInput";   // Oil separator stage 2 oil return pressure
      HBL_CT_643 { S7_SetPoint := 'True'} : "stAnalogInput";   // Gas detector suction accumulator popoff
      HBL_LT_650 { S7_SetPoint := 'True'} : "stAnalogInput";   // Heat source condensate buffer tank level
      HBL_CT_673 { S7_SetPoint := 'True'} : "stAnalogInput";   // Gas detector oil separator discharge popoff
      HBL_PT_651 { S7_SetPoint := 'True'} : "stAnalogInput";   // Heat source condensate buffer tank pressure
      HBL_PT_701 { S7_SetPoint := 'True'} : "stAnalogInput";   // Filter dryer suction pressure
      HBL_PT_702 { S7_SetPoint := 'True'} : "stAnalogInput";   // Filter dryer discharge pressure
      HBL_PT_703 { S7_SetPoint := 'True'} : "stAnalogInput";   // Filter dryer differential pressure
      CPC_CT_851 { S7_SetPoint := 'True'} : "stAnalogInput";   // Gas detector CPC popoff
      CPC_PT_862 { S7_SetPoint := 'True'} : "stAnalogInput";   // CPC pump discharge pressure
      CPC_PT_865 { S7_SetPoint := 'True'} : "stAnalogInput";   // CPC pump suction pressure
      CPC_TT_866 { S7_SetPoint := 'True'} : "stAnalogInput";   // CPC pump suction temperature
      CPC_LT_870 { S7_SetPoint := 'True'} : "stAnalogInput";   // CPC tank refrigerant level
      CPC_TT_871 { S7_SetPoint := 'True'} : "stAnalogInput";   // CPC tank refrigerant temperature
      CPC_PT_872 { S7_SetPoint := 'True'} : "stAnalogInput";   // CPC tank refrigerant pressure
      HBL_TT_901 { S7_SetPoint := 'True'} : "stAnalogInput";   // Heat sink suction temperature
      HBL_PT_902 { S7_SetPoint := 'True'} : "stAnalogInput";   // Heat sink suction pressure
      HBL_TT_03 { S7_SetPoint := 'True'} : "stAnalogInput";   // Oil sump oil temperature
      HBL_TT_16 { S7_SetPoint := 'True'} : "stAnalogInput";   // Container air temperature
      HBL_TT_17 { S7_SetPoint := 'True'} : "stAnalogInput";   // Control cabinet air temperature
      HBL_TT_18 { S7_SetPoint := 'True'} : "stAnalogInput";   // Ambient air temperature
      HBL_TT_20 { S7_SetPoint := 'True'} : "stAnalogInput";   // Compressor motor winding temperature
      HBL_TT_21 { S7_SetPoint := 'True'} : "stAnalogInput";   // Oil sump wall temperature left
      HBL_TT_22 { S7_SetPoint := 'True'} : "stAnalogInput";   // Oil sump wall temperature right
      HBL_TT_23 { S7_SetPoint := 'True'} : "stAnalogInput";   // Compressor motor U-winding temperature
      HBL_TT_24 { S7_SetPoint := 'True'} : "stAnalogInput";   // Compressor motor V-winding temperature
      HBL_TT_25 { S7_SetPoint := 'True'} : "stAnalogInput";   // Compressor motor W-winding temperature
      HBL_TT_26 { S7_SetPoint := 'True'} : "stAnalogInput";   // Compressor motor D bearing temperature
      HBL_TT_27 { S7_SetPoint := 'True'} : "stAnalogInput";   // Compressor motor N bearing temperature
      HBL_PT_05 { S7_SetPoint := 'True'} : "stAnalogInput";   // Crankcase gas pressure
      HBL_PT_960 { S7_SetPoint := 'True'} : "stAnalogInput";   // Oil pump discharge pressure
      HBL_PT_961 { S7_SetPoint := 'True'} : "stAnalogInput";   // Oil gallery pressure
      HBL_CT_01 { S7_SetPoint := 'True'} : "stAnalogInput";   // Gas detector Heatbooster (optional)
      HBL_CT_950 { S7_SetPoint := 'True'} : "stAnalogInput";   // Gas detector container/compressor room
      SSC_TT_01 { S7_SetPoint := 'True'} : "stAnalogInput";   // SSC seal suction temperature
      SSC_TT_02 { S7_SetPoint := 'True'} : "stAnalogInput";   // SSC seal discharge temperature
      SSC_TT_03 { S7_SetPoint := 'True'} : "stAnalogInput";   // SSC barrier fluid circulation pump suction temperature
      SSC_TT_04 { S7_SetPoint := 'True'} : "stAnalogInput";   // SSC barrier fluid heat exchanger temperature
      SSC_PIT_01 { S7_SetPoint := 'True'} : "stAnalogInput";   // SSC barrier fluid accumulator pressure
      SSC_PDT_01 { S7_SetPoint := 'True'} : "stAnalogInput";   // SSC barrier fluid circulation pump differential pressure
      SSC_LT_01 { S7_SetPoint := 'True'} : "stAnalogInput";   // SSC barrier fluid reservoir level
      Spare { S7_SetPoint := 'True'} : "stAnalogInput";
   END_VAR
BEGIN
   HBL_TT_502.Raw.iMin := -14500;
   HBL_TT_502.Raw.iMax := 15500;
   HBL_TT_502.Eng.fMin := -145.0;
   HBL_TT_502.Eng.fMax := 155.0;
   HBL_PT_503.Raw.iMin := 0;
   HBL_PT_503.Raw.iMax := 27648;
   HBL_PT_503.Eng.fMin := 0.0;
   HBL_PT_503.Eng.fMax := 6000.0;
   HBL_TT_504.Raw.iMin := -14500;
   HBL_TT_504.Raw.iMax := 15500;
   HBL_TT_504.Eng.fMin := -145.0;
   HBL_TT_504.Eng.fMax := 155.0;
   HBL_TT_505.Raw.iMin := -14500;
   HBL_TT_505.Raw.iMax := 15500;
   HBL_TT_505.Eng.fMin := -145.0;
   HBL_TT_505.Eng.fMax := 155.0;
   HBL_PT_506.Eng.fMin := 0.0;
   HBL_PT_506.Eng.fMax := 2500.0;
   HBL_LT_510.Raw.iMin := 0;
   HBL_LT_510.Raw.iMax := 27648;
   HBL_LT_510.Eng.fMin := 0.0;
   HBL_LT_510.Eng.fMax := 100.0;
   HBL_PT_511.Raw.iMin := 0;
   HBL_PT_511.Raw.iMax := 27648;
   HBL_PT_511.Eng.fMin := 0.0;
   HBL_PT_511.Eng.fMax := 4000.0;
   HBL_TT_512.Raw.iMin := -14500;
   HBL_TT_512.Raw.iMax := 15500;
   HBL_TT_512.Eng.fMin := -145.0;
   HBL_TT_512.Eng.fMax := 155.0;
   HBL_TT_516.Raw.iMin := -14500;
   HBL_TT_516.Raw.iMax := 15500;
   HBL_TT_516.Eng.fMin := -145.0;
   HBL_TT_516.Eng.fMax := 155.0;
   HBL_PT_517.Raw.iMin := 0;
   HBL_PT_517.Raw.iMax := 27648;
   HBL_PT_517.Eng.fMax := 4000.0;
   HBL_TT_518.Raw.iMin := -14500;
   HBL_TT_518.Raw.iMax := 15500;
   HBL_TT_518.Eng.fMin := -145.0;
   HBL_TT_518.Eng.fMax := 155.0;
   HBL_PT_519.Raw.iMax := 27648;
   HBL_PT_519.Eng.fMax := 2500.0;
   HBL_FT_520.Raw.iMin := 0;
   HBL_FT_520.Raw.iMax := 27648;
   HBL_FT_520.Eng.fMin := 0.0;
   HBL_FT_520.Eng.fMax := 16.667;
   // HBL_FT_520.Eng.fValue : [L/s]
   HBL_CT_524.Eng.fMin := 0.0;
   HBL_CT_524.Eng.fMax := 5000.0;
   HBL_TT_525.Raw.iMin := -14500;
   HBL_TT_525.Raw.iMax := 15500;
   HBL_TT_525.Eng.fMin := -145.0;
   HBL_TT_525.Eng.fMax := 155.0;
   HBL_PT_526.Raw.iMax := 27648;
   HBL_PT_526.Eng.fMax := 4000.0;
   HBL_TT_530.Raw.iMin := -14500;
   HBL_TT_530.Raw.iMax := 15500;
   HBL_TT_530.Eng.fMin := -145.0;
   HBL_TT_530.Eng.fMax := 155.0;
   HBL_PT_531.Raw.iMin := 0;
   HBL_PT_531.Raw.iMax := 27648;
   HBL_PT_531.Eng.fMin := 0.0;   // [kPa]
   HBL_PT_531.Eng.fMax := 3450.0;   // [kPa]
   HBL_TT_532.Raw.iMin := -14500;
   HBL_TT_532.Raw.iMax := 15500;
   HBL_TT_532.Eng.fMin := -145.0;
   HBL_TT_532.Eng.fMax := 155.0;
   HBL_TT_533.Raw.iMin := -14500;
   HBL_TT_533.Raw.iMax := 15500;
   HBL_TT_533.Eng.fMin := -145.0;
   HBL_TT_533.Eng.fMax := 155.0;
   HBL_PT_534.Raw.iMin := 0;
   HBL_PT_534.Raw.iMax := 27648;
   HBL_PT_534.Eng.fMin := 0.0;   // [kPa]
   HBL_PT_534.Eng.fMax := 3450.0;   // [kPa]
   HBL_AT_535.Raw.iMin := 0;
   HBL_AT_535.Raw.iMax := 27648;
   HBL_AT_535.Eng.fMin := 0.84;
   HBL_AT_535.Eng.fMax := 1.05;
   HBL_CT_538.Eng.fMin := 0.0;
   HBL_CT_538.Eng.fMax := 5000.0;
   HBL_TT_540.Raw.iMin := -14500;
   HBL_TT_540.Raw.iMax := 15500;
   HBL_TT_540.Eng.fMin := -145.0;
   HBL_TT_540.Eng.fMax := 155.0;
   HBL_PT_541.Raw.iMin := 0;
   HBL_PT_541.Raw.iMax := 27648;
   HBL_PT_541.Eng.fMin := 0.0;   // [kPa]
   HBL_PT_541.Eng.fMax := 3450.0;   // [kPa]
   HBL_TT_542.Raw.iMin := -14500;
   HBL_TT_542.Raw.iMax := 15500;
   HBL_TT_542.Eng.fMin := -145.0;
   HBL_TT_542.Eng.fMax := 155.0;
   HBL_TT_543.Raw.iMin := -14500;
   HBL_TT_543.Raw.iMax := 15500;
   HBL_TT_543.Eng.fMin := -145.0;
   HBL_TT_543.Eng.fMax := 155.0;
   HBL_PT_544.Raw.iMax := 27648;
   HBL_PT_544.Eng.fMin := 0.0;   // [kPa]
   HBL_PT_544.Eng.fMax := 3450.0;   // [kPa]
   HBL_AT_545.Raw.iMin := 0;
   HBL_AT_545.Raw.iMax := 27648;
   HBL_AT_545.Eng.fMin := 0.84;
   HBL_AT_545.Eng.fMax := 1.05;
   HBL_TT_546.Raw.iMin := -14500;
   HBL_TT_546.Raw.iMax := 15500;
   HBL_TT_546.Eng.fMin := -145.0;
   HBL_TT_546.Eng.fMax := 155.0;
   HBL_PT_547.Raw.iMin := 0;
   HBL_PT_547.Raw.iMax := 27648;
   HBL_PT_547.Eng.fMin := 0.0;
   HBL_PT_547.Eng.fMax := 2500.0;
   HBL_PT_561.Eng.fMin := 0.0;
   HBL_PT_561.Eng.fMax := 200.0;
   HBL_PT_562.Eng.fMin := 0.0;
   HBL_PT_562.Eng.fMax := 200.0;
   HBL_FT_565.Eng.fMin := 0.0;
   HBL_FT_565.Eng.fMax := 100.0;
   HBL_FT_566.Eng.fMin := 0.0;
   HBL_FT_566.Eng.fMax := 100.0;
   HBL_TT_571.Raw.iMin := -14500;
   HBL_TT_571.Raw.iMax := 15500;
   HBL_TT_571.Eng.fMin := -145.0;
   HBL_TT_571.Eng.fMax := 155.0;
   HBL_PT_572.Raw.iMin := 0;
   HBL_PT_572.Raw.iMax := 27648;
   HBL_PT_572.Eng.fMin := 0.0;
   HBL_PT_572.Eng.fMax := 4000.0;
   HBL_TT_573.Raw.iMin := -14500;
   HBL_TT_573.Raw.iMax := 15500;
   HBL_TT_573.Eng.fMin := -145.0;
   HBL_TT_573.Eng.fMax := 155.0;
   HBL_PT_580.Eng.fMin := 0.0;
   HBL_PT_580.Eng.fMax := 4000.0;
   HBL_LT_610.Raw.iMin := 0;
   HBL_LT_610.Raw.iMax := 27648;
   HBL_LT_610.Eng.fMin := 0.0;
   HBL_LT_610.Eng.fMax := 100.0;
   HBL_TT_611.Raw.iMin := -14500;
   HBL_TT_611.Raw.iMax := 15500;
   HBL_TT_611.Eng.fMin := -145.0;
   HBL_TT_611.Eng.fMax := 155.0;
   HBL_PT_612.Raw.iMax := 27648;
   HBL_PT_612.Eng.fMax := 4000.0;
   HBL_CT_615.Raw.iMin := 0;
   HBL_CT_615.Raw.iMax := 27648;
   HBL_CT_615.Eng.fMin := 0.0;
   HBL_CT_615.Eng.fMax := 2000.0;
   HBL_PT_618.Raw.iMin := 0;
   HBL_PT_618.Raw.iMax := 27648;
   HBL_PT_618.Eng.fMin := 0.0;
   HBL_PT_618.Eng.fMax := 3450.0;
   HBL_CT_620.Eng.fMin := 0.0;
   HBL_CT_620.Eng.fMax := 5000.0;
   HBL_PT_635.Raw.iMin := 0;
   HBL_PT_635.Raw.iMax := 27648;
   HBL_PT_635.Eng.fMin := 0.0;   // [kPa]
   HBL_PT_635.Eng.fMax := 3450.0;   // [kPa]
   HBL_PT_636.Raw.iMin := 0;
   HBL_PT_636.Raw.iMax := 27648;
   HBL_PT_636.Eng.fMin := 0.0;   // [kPa]
   HBL_PT_636.Eng.fMax := 3450.0;   // [kPa]
   HBL_CT_643.Eng.fMin := 0.0;
   HBL_CT_643.Eng.fMax := 5000.0;
   HBL_LT_650.Raw.iMin := 0;
   HBL_LT_650.Raw.iMax := 27648;
   HBL_LT_650.Eng.fMin := 0.0;
   HBL_LT_650.Eng.fMax := 100.0;
   HBL_CT_673.Eng.fMin := 0.0;
   HBL_CT_673.Eng.fMax := 5000.0;
   HBL_PT_651.Raw.iMin := 0;
   HBL_PT_651.Raw.iMax := 27648;
   HBL_PT_651.Eng.fMin := -10.0;   // [kPa]
   HBL_PT_651.Eng.fMax := 1000.0;   // [kPa]
   HBL_PT_701.Raw.iMin := 0;
   HBL_PT_701.Raw.iMax := 27648;
   HBL_PT_701.Eng.fMin := 0.0;
   HBL_PT_701.Eng.fMax := 3450.0;
   HBL_PT_702.Raw.iMin := 0;
   HBL_PT_702.Raw.iMax := 27648;
   HBL_PT_702.Eng.fMin := 0.0;
   HBL_PT_702.Eng.fMax := 3450.0;
   CPC_CT_851.Eng.fMin := 0.0;
   CPC_CT_851.Eng.fMax := 5000.0;
   CPC_PT_862.Raw.iMax := 27648;
   CPC_PT_862.Eng.fMin := 0.0;
   CPC_PT_862.Eng.fMax := 6000.0;
   CPC_PT_865.Eng.fMin := 0.0;
   CPC_PT_865.Eng.fMax := 1600.0;
   CPC_TT_866.Raw.iMin := -14500;
   CPC_TT_866.Raw.iMax := 15500;
   CPC_TT_866.Eng.fMin := -145.0;
   CPC_TT_866.Eng.fMax := 155.0;
   CPC_LT_870.Raw.iMax := 27648;
   CPC_LT_870.Eng.fMax := 100.0;
   CPC_TT_871.Raw.iMin := -14500;
   CPC_TT_871.Raw.iMax := 15500;
   CPC_TT_871.Eng.fMin := -145.0;
   CPC_TT_871.Eng.fMax := 155.0;
   CPC_PT_872.Raw.iMin := 0;
   CPC_PT_872.Raw.iMax := 27648;
   CPC_PT_872.Eng.fMin := 0.0;
   CPC_PT_872.Eng.fMax := 3450.0;
   HBL_TT_901.Raw.iMin := -14500;
   HBL_TT_901.Raw.iMax := 15500;
   HBL_TT_901.Eng.fMin := -145.0;
   HBL_TT_901.Eng.fMax := 155.0;
   HBL_PT_902.Raw.iMin := 0;
   HBL_PT_902.Raw.iMax := 27648;
   HBL_PT_902.Eng.fMin := 0.0;
   HBL_PT_902.Eng.fMax := 2500.0;
   HBL_TT_03.Raw.iMin := -14500;
   HBL_TT_03.Raw.iMax := 15500;
   HBL_TT_03.Eng.fMin := -145.0;
   HBL_TT_03.Eng.fMax := 155.0;
   HBL_TT_16.Raw.iMin := -14500;
   HBL_TT_16.Raw.iMax := 15500;
   HBL_TT_16.Eng.fMin := -145.0;
   HBL_TT_16.Eng.fMax := 155.0;
   HBL_TT_17.Raw.iMin := -14500;
   HBL_TT_17.Raw.iMax := 15500;
   HBL_TT_17.Eng.fMin := -145.0;
   HBL_TT_17.Eng.fMax := 155.0;
   HBL_TT_18.Raw.iMin := -14500;
   HBL_TT_18.Raw.iMax := 15500;
   HBL_TT_18.Eng.fMin := -145.0;
   HBL_TT_18.Eng.fMax := 155.0;
   HBL_TT_20.Raw.iMin := -14500;
   HBL_TT_20.Raw.iMax := 15500;
   HBL_TT_20.Eng.fMin := -145.0;
   HBL_TT_20.Eng.fMax := 155.0;
   HBL_TT_21.Raw.iMin := -14500;
   HBL_TT_21.Raw.iMax := 15500;
   HBL_TT_21.Eng.fMin := -145.0;
   HBL_TT_21.Eng.fMax := 155.0;
   HBL_TT_22.Raw.iMin := -14500;
   HBL_TT_22.Raw.iMax := 15500;
   HBL_TT_22.Eng.fMin := -145.0;
   HBL_TT_22.Eng.fMax := 155.0;
   HBL_TT_23.Raw.iMin := -14500;
   HBL_TT_23.Raw.iMax := 15500;
   HBL_TT_23.Eng.fMin := -145.0;
   HBL_TT_23.Eng.fMax := 155.0;
   HBL_TT_24.Raw.iMin := -14500;
   HBL_TT_24.Raw.iMax := 15500;
   HBL_TT_24.Eng.fMin := -145.0;
   HBL_TT_24.Eng.fMax := 155.0;
   HBL_TT_25.Raw.iMin := -14500;
   HBL_TT_25.Raw.iMax := 15500;
   HBL_TT_25.Eng.fMin := -145.0;
   HBL_TT_25.Eng.fMax := 155.0;
   HBL_TT_26.Raw.iMin := -14500;
   HBL_TT_26.Raw.iMax := 15500;
   HBL_TT_26.Eng.fMin := -145.0;
   HBL_TT_26.Eng.fMax := 155.0;
   HBL_TT_27.Raw.iMin := -14500;
   HBL_TT_27.Raw.iMax := 15500;
   HBL_TT_27.Eng.fMin := -145.0;
   HBL_TT_27.Eng.fMax := 155.0;
   HBL_PT_05.Raw.iMax := 27648;
   HBL_PT_05.Eng.fMax := 2500.0;
   HBL_PT_960.Raw.iMax := 27648;
   HBL_PT_960.Eng.fMax := 2500.0;
   HBL_PT_961.Raw.iMin := 0;
   HBL_PT_961.Raw.iMax := 27648;
   HBL_PT_961.Eng.fMin := 0.0;
   HBL_PT_961.Eng.fMax := 2500.0;
   HBL_CT_01.Raw.iMin := 0;
   HBL_CT_01.Raw.iMax := 27648;
   HBL_CT_01.Eng.fMin := 0.0;
   HBL_CT_01.Eng.fMax := 5000.0;
   HBL_CT_950.Raw.iMin := 0;
   HBL_CT_950.Raw.iMax := 27648;
   HBL_CT_950.Eng.fMin := 0.0;
   HBL_CT_950.Eng.fMax := 2000.0;
   SSC_TT_01.Raw.iMin := -14500;
   SSC_TT_01.Raw.iMax := 15500;
   SSC_TT_01.Eng.fMin := -145.0;
   SSC_TT_01.Eng.fMax := 155.0;
   SSC_TT_02.Raw.iMin := -14500;
   SSC_TT_02.Raw.iMax := 15500;
   SSC_TT_02.Eng.fMin := -145.0;
   SSC_TT_02.Eng.fMax := 155.0;
   SSC_TT_03.Raw.iMin := -14500;
   SSC_TT_03.Raw.iMax := 15500;
   SSC_TT_03.Eng.fMin := -145.0;
   SSC_TT_03.Eng.fMax := 155.0;
   SSC_TT_04.Raw.iMin := -14500;
   SSC_TT_04.Raw.iMax := 15500;
   SSC_TT_04.Eng.fMin := -145.0;
   SSC_TT_04.Eng.fMax := 155.0;
   SSC_PIT_01.Raw.iMin := 0;
   SSC_PIT_01.Raw.iMax := 27648;
   SSC_PIT_01.Eng.fMin := 0.0;
   SSC_PIT_01.Eng.fMax := 2500.0;
   SSC_PDT_01.Raw.iMin := 0;
   SSC_PDT_01.Raw.iMax := 27648;
   SSC_PDT_01.Eng.fMin := 0.0;
   SSC_PDT_01.Eng.fMax := 250.0;
   SSC_LT_01.Raw.iMin := 0;
   SSC_LT_01.Raw.iMax := 27648;
   SSC_LT_01.Eng.fMin := 0.0;
   SSC_LT_01.Eng.fMax := 100.0;
END_DATA_BLOCK

DATA_BLOCK "DB_AO"   // DB5
{ S7_Optimized_Access := 'TRUE' }
AUTHOR : Heaten
VERSION : 0.1
// stored: AutoNumber true, DBAccessibleFromOPCUA true, DBAccessibleFromWebserver true, IsOnlyStoredInLoadMemory false, IsRetainMemResEnabled false, IsWriteProtectedInAS false, MemoryReserve 100
BEGIN
END_DATA_BLOCK

